// TIA Portal V20 export
VAR_GLOBAL   // PLC tag table "IMC84"
   "IMC84Sensor -1" AT %I583.0 : Bool;   // High = Sensor active (input type and polarity can be configured)
   IMC84Sensor_2 AT %I583.1 : Bool;   // High = Sensor active (input type and polarity can be configured)
   IMC84Sensor_3 AT %I583.2 : Bool;   // High = Sensor active (input type and polarity can be configured)
   IMC84Sensor_4 AT %I583.3 : Bool;   // High = Sensor active (input type and polarity can be configured)
   IMC84Sensor_5 AT %I583.4 : Bool;
   IMC84Sensor_6 AT %I583.5 : Bool;
   IMC84Sensor_7 AT %I583.6 : Bool;
   IMC84Sensor_8 AT %I583.7 : Bool;
   IMC84IO1 AT %I584.0 : Bool;   // Digital I/O PLC Input PLC Output
   IMC84IO2 AT %I584.1 : Bool;   // Digital I/O PLC Input PLC Output
   IMC84IO3 AT %I584.2 : Bool;   // Digital I/O PLC Input PLC Output
   IMC84IO4 AT %I584.3 : Bool;   // Digital I/O PLC Input PLC Output
   IMC84IO5 AT %I584.4 : Bool;
   IMC84IO6 AT %I584.5 : Bool;
   IMC84IO7 AT %I584.6 : Bool;
   IMC84IO8 AT %I584.7 : Bool;
   "IMC84MotorStateErrorRD -G1.4.3" AT %I585.0 : Bool;   // High = Motor Error; Low = Motor OK
   "IMC84MotorStateErrorRD -G1.4.2" AT %I585.1 : Bool;   // High = Motor Error; Low = Motor OK
   "IMC84MotorStateErrorRD -G1.4.1" AT %I585.2 : Bool;   // High = Motor Error; Low = Motor OK
   "IMC84MotorStateErrorRD_G1.3.1" AT %I585.3 : Bool;   // High = Motor Error; Low = Motor OK
   "IMC84MotorStateSpeedRD -G1.4.3" AT %IB586 : SInt;   // Speed 0–100 ( 0 = Stop, 100 = max speed), negative sign reverses the turning direction
   "IMC84MotorStateSpeedRD -G1.4.2" AT %IB587 : SInt;   // Speed 0–100 ( 0 = Stop, 100 = max speed), negative sign reverses the turning direction
   "IMC84MotorStateSpeedRD -G1.4.1" AT %IB588 : SInt;   // Speed 0–100 ( 0 = Stop, 100 = max speed), negative sign reverses the turning direction
   "IMC84MotorStateSpeedRD_G1.3.1" AT %IB589 : SInt;   // Speed 0–100 ( 0 = Stop, 100 = max speed), negative sign reverses the turning direction
   "IMC84MotorCurrentRD -G1.4.3" AT %IW591 : Int;   // Average current in mA
   "IMC84MotorCurrentRD -G1.4.2" AT %IW593 : Int;   // Average current in mA
   "IMC84MotorCurrentRD -G1.4.1" AT %IW595 : Int;   // Average current in mA
   "IMC84MotorCurrentRD_G1.3.1" AT %IW597 : Int;   // Average current in mA
   "IMC84Voltage(MotorPower)" AT %IW599 : Int;   // Voltage „Motor Power“ in mV
   "IMC84Voltage(Sensors)" AT %IW601 : Int;   // Voltage „Power Logic + Sensors“ in mV
   IMC84Temperature AT %IW603 : Int;   // Temperature in 0,1 C
   IMC84SystemUpTime AT %ID605 : DInt;   // Operating time in seconds since the last start/restart
   "IMC84DigitalOutputRD -G1.4.3" AT %Q64.0 : Bool;
   "IMC84DigitalOutputRD -G1.4.2" AT %Q64.1 : Bool;
   "IMC84DigitalOutputRD -G1.4.1" AT %Q64.2 : Bool;
   "IMC84DigitalOutputRD_G1.3.1" AT %Q64.3 : Bool;
   "IMC84MotorTargetSpeedRD -G1.4.3" AT %QB65 : SInt;   // Speed 0–100 ( 0 = Stop, 100 = max speed), negative sign reverses the turning direction
   "IMC84MotorTargetSpeedRD -G1.4.2" AT %QB66 : SInt;   // Speed 0–100 ( 0 = Stop, 100 = max speed), negative sign reverses the turning direction
   "IMC84MotorTargetSpeedRD -G1.4.1" AT %QB67 : SInt;   // Speed 0–100 ( 0 = Stop, 100 = max speed), negative sign reverses the turning direction
   "IMC84MotorTargetSpeedRD_G1.3.1" AT %QB68 : SInt;   // Speed 0–100 ( 0 = Stop, 100 = max speed), negative sign reverses the turning direction
END_VAR
